//{attribute 'qualified_only'}
VAR_GLOBAL

	
END_VAR

(* stored: Version 1.1.0.1, ProductVersion 3.1.4024.6
   GVL Main: Id {743c36cb-e5dd-4408-91ed-5169699d82d2} *)
